(* CoDeSys 2.3 export: WORD_TO_VAR.EXP *)

(* POU FUNv1/WORD_TO_VAR, ST *)
FUNCTION WORD_TO_VAR : VarST
VAR_IN_OUT
    in : WORD;
END_VAR
VAR
END_VAR
WORD_TO_VAR.pby   := ADR(in);
WORD_TO_VAR.type_ := WORD_;
END_FUNCTION
